(* CoDeSys 2.3 export: UUID.EXP *)

(* Data type *)
TYPE UUID : ARRAY[0..15] OF BYTE;
END_TYPE
